TYPE EcCoeSdoRead_Status_typ :
	STRUCT
		bBusy           : BOOL;
        bError          : BOOL;
	END_STRUCT
END_TYPE

(* stored: Version 1.1.0.1, ProductVersion 3.1.4024.3
   DUT EcCoeSdoRead_Status_typ: Id {5fbdc19e-9ea9-0e23-1e5c-4da9a1fb26b3} *)
